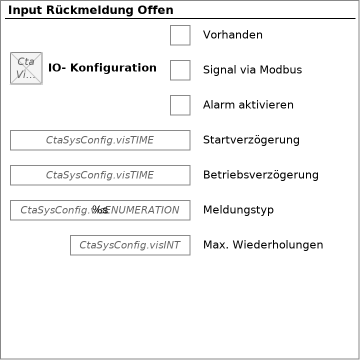
VISUALIZATION StellAntrieb_ParameterIO2  // 360x360
VAR_INPUT
    ITF_STELLANTRIEBIN 	:	ITF_STELLANTRIEB;
	ITF_RückOffen_IN	:	CtaSysIO.ITF_IO;
END_VAR
    Label (5,0 350x20), "Input Rückmeldung Offen"
    Frame (170,25 20x20)
        shows CtaSysConfig.visBOOL(visfbBOOLIn := ITF_STELLANTRIEBIN.p_scInStellAtRükOpen_fbxEnable)
    Label (200,25 150x20), "Vorhanden"
    Frame (170,60 20x20)
        shows CtaSysConfig.visBOOL(visfbBOOLIn := ITF_STELLANTRIEBIN.p_scInStellAtRükOpen_fbxInputMb)
    Label (200,60 150x20), "Signal via Modbus"
    Frame (170,95 20x20)
        shows CtaSysConfig.visBOOL(visfbBOOLIn := ITF_STELLANTRIEBIN.p_scInStellAtRükOpen_fbxDoesAlarm)
    Label (200,95 150x20), "Alarm aktivieren"
    Frame (10,130 180x20)
        shows CtaSysConfig.visTIME(visfbTIMEIn := ITF_STELLANTRIEBIN.p_scInStellAtRükOpen_fbtDelayStart)
    Label (200,130 150x20), "Startverzögerung"
    Label (200,165 150x20), "Betriebsverzögerung"
    Frame (10,165 180x20)
        shows CtaSysConfig.visTIME(visfbTIMEIn := ITF_STELLANTRIEBIN.p_scInStellAtRükOpen_fbtDelayRun)
    Label (200,200 150x20), "Meldungstyp"
    Label (200,235 150x20), "Max. Wiederholungen"
    Line (5,18) (355,18)
    Frame (10,200 180x20)
        shows CtaSysConfig.visENUMERATION(visfbENUIn := ITF_STELLANTRIEBIN.p_scInStellAtRükOpen_fbiTypeOfAck)
    Frame (70,235 120x20)
        shows CtaSysConfig.visINT(visfbINTIn := ITF_STELLANTRIEBIN.p_scInStellAtRükOpen_fbiMaxErrorRetryAllowed)
    Image (10,52 32x32), invisible if: ITF_RückOffen_IN = 0, image: CtaVisSymbols.ImagePool.build
        OnMouseDown:  Dialog=StellAntrieb_POPUP_IO_ITF, Parameters={ITF_IO_IN: ITF_RückOffen_IN}, OpenModal=True, OpenCentered=True
    Label (45,58 120x20), "IO- Konfiguration", invisible if: ITF_RückOffen_IN = 0
    Textfield (30,200 140x20), "%s", text list: 'CtaAppReport.txtLibAp99_2enTypeOfAck', text index: CtaSysConfig.fcGetEnumerationId(ITF_STELLANTRIEBIN.p_scInStellAtRükOpen_fbiTypeOfAck)
END_VISUALIZATION

// 40 Visualizations/POPUP/PARAMETER/StellAntrieb_IO/StellAntrieb_ParameterIO3
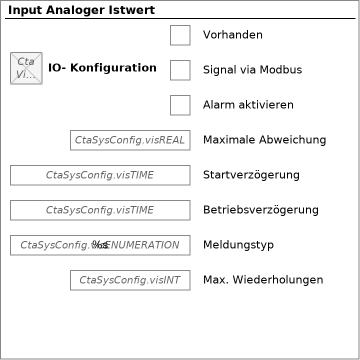
VISUALIZATION StellAntrieb_ParameterIO3  // 360x360
VAR_INPUT
    ITF_STELLANTRIEBIN 	:	ITF_STELLANTRIEB;
	ITF_ActualPos_IN	:	CtaSysIO.ITF_IO;
END_VAR
    Label (5,0 350x20), "Input Analoger Istwert"
    Frame (170,25 20x20)
        shows CtaSysConfig.visBOOL(visfbBOOLIn := ITF_STELLANTRIEBIN.p_scInStellAtActualPosition_fbxEnable)
    Label (200,25 150x20), "Vorhanden"
    Frame (170,60 20x20)
        shows CtaSysConfig.visBOOL(visfbBOOLIn := ITF_STELLANTRIEBIN.p_scInStellAtActualPosition_fbxInputMb)
    Label (200,60 150x20), "Signal via Modbus"
    Frame (170,95 20x20)
        shows CtaSysConfig.visBOOL(visfbBOOLIn := ITF_STELLANTRIEBIN.p_scInStellAtActualPosition_fbxDoesAlarm)
    Label (200,95 150x20), "Alarm aktivieren"
    Frame (10,165 180x20)
        shows CtaSysConfig.visTIME(visfbTIMEIn := ITF_STELLANTRIEBIN.p_scInStellAtActualPosition_fbtDelayStart)
    Label (200,165 150x20), "Startverzögerung"
    Label (200,200 150x20), "Betriebsverzögerung"
    Frame (10,200 180x20)
        shows CtaSysConfig.visTIME(visfbTIMEIn := ITF_STELLANTRIEBIN.p_scInStellAtActualPosition_fbtDelayRun)
    Frame (70,130 120x20)
        shows CtaSysConfig.visREAL(visfbREALIn := ITF_STELLANTRIEBIN.p_scInStellAtActualPosition_fbrMaxDiff, stPhysikalischeEinheit := '%')
    Label (200,130 150x20), "Maximale Abweichung"
    Label (200,235 150x20), "Meldungstyp"
    Label (200,270 150x20), "Max. Wiederholungen"
    Line (5,18) (355,18)
    Frame (10,235 180x20)
        shows CtaSysConfig.visENUMERATION(visfbENUIn := ITF_STELLANTRIEBIN.p_scInStellAtActualPosition_fbiTypeOfAck)
    Frame (70,270 120x20)
        shows CtaSysConfig.visINT(visfbINTIn := ITF_STELLANTRIEBIN.p_scInStellAtActualPosition_fbiMaxErrorRetryAllowed)
    Label (45,58 120x20), "IO- Konfiguration", invisible if: ITF_ActualPos_IN = 0
    Image (10,52 32x32), invisible if: ITF_ActualPos_IN = 0, image: CtaVisSymbols.ImagePool.build
        OnMouseDown:  Dialog=StellAntrieb_POPUP_IO_ITF, Parameters={ITF_IO_IN: ITF_ActualPos_IN}, OpenModal=True, OpenCentered=True
    Textfield (30,235 140x20), "%s", text list: 'CtaAppReport.txtLibAp99_2enTypeOfAck', text index: CtaSysConfig.fcGetEnumerationId(ITF_STELLANTRIEBIN.p_scInStellAtActualPosition_fbiTypeOfAck)
END_VISUALIZATION

// 40 Visualizations/POPUP/PARAMETER/StellAntrieb_InfluxDb/StellAntrieb_ParameterInfluxDb
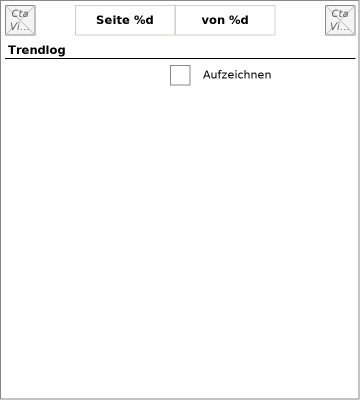
VISUALIZATION StellAntrieb_ParameterInfluxDb  // 360x400
VAR_INPUT
    ITF_STELLANTRIEBIN : ITF_STELLANTRIEB;
END_VAR
VAR
    uiPage  :   UINT;
    uiMin   :   UINT    := 0;
    uiMax   :   UINT    := 0;
END_VAR
    Image (5,5 30x30), invisible if: uiPage = uiMin, image: CtaVisSymbols.ImagePool.arrow-left_square
        OnMouseClick: execute {
            uiPage := uiPage - 1;
            IF uiPage <= uiMin THEN
                uiPage := uiMin;
            END_IF;
        }
    Image (325,5 30x30), invisible if: uiPage = uiMax, image: CtaVisSymbols.ImagePool.arrow-right_square
        OnMouseClick: execute {
            uiPage := uiPage + 1;
            IF uiPage >= uiMax THEN
                uiPage := uiMax;
            END_IF;
        }
    Frame (0,40 360x360), frame switch variable: uiPage
        shows StellAntrieb_ParameterInfluxDb0(ITF_STELLANTRIEBIN := ITF_STELLANTRIEBIN)
        shows AT_ParameterIO1(ITF_Parameter := ITF_Parameter)
        pReferences[0]: ITF_Parameter=ITF_Parameter
    Textfield (75,5 100x30), "Seite %d", text variable: uiPage
    Textfield (175,5 100x30), "von %d", text variable: uiMax
END_VISUALIZATION

// 40 Visualizations/POPUP/PARAMETER/StellAntrieb_InfluxDb/StellAntrieb_ParameterInfluxDb0
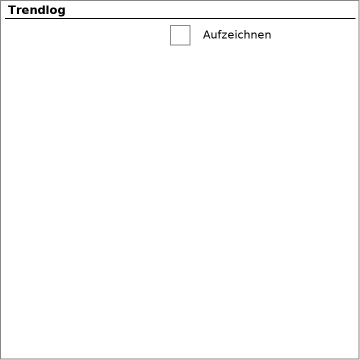
VISUALIZATION StellAntrieb_ParameterInfluxDb0  // 360x360
VAR_INPUT
    ITF_STELLANTRIEBIN : ITF_STELLANTRIEB;
END_VAR
    Frame (170,25 20x20)
        shows CtaSysConfig.visBOOL(visfbBOOLIn := ITF_STELLANTRIEBIN.p_scInfluxDb_fbxEnable)
    Label (200,25 150x20), "Aufzeichnen"
    Label (5,0 350x20), "Trendlog"
    Line (5,18) (355,18)
END_VISUALIZATION

// 40 Visualizations/POPUP/IO/StellAntrieb_IO0
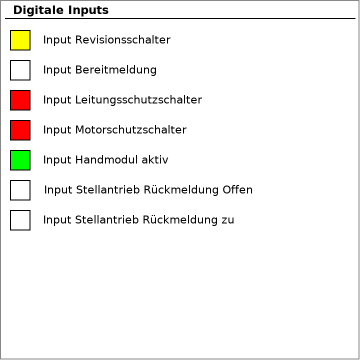
VISUALIZATION StellAntrieb_IO0  // 360x360
VAR_INPUT
    ITF_STELLANTRIEBIN    :   ITF_STELLANTRIEB;	
END_VAR
    Label (40,30 320x20), "Input Revisionsschalter", invisible if: ITF_STELLANTRIEBIN.proNotShowDI_RevisionSwitchOk
    Label (40,60 320x20), "Input Bereitmeldung", invisible if: ITF_STELLANTRIEBIN.proNotShowDI_Ready
    Rectangle (10,30 20x20), colour toggle: ITF_STELLANTRIEBIN.proGetDI_RevisionSwitchOK, invisible if: ITF_STELLANTRIEBIN.proNotShowDI_RevisionSwitchOk
    Rectangle (10,60 20x20), colour toggle: ITF_STELLANTRIEBIN.proGetDI_IsReady, invisible if: ITF_STELLANTRIEBIN.proNotShowDI_Ready
    Rectangle (10,90 20x20), colour toggle: ITF_STELLANTRIEBIN.proGetDI_FuseOK, invisible if: ITF_STELLANTRIEBIN.proNotShowDI_FuseOk
    Label (40,90 320x20), "Input Leitungsschutzschalter", invisible if: ITF_STELLANTRIEBIN.proNotShowDI_FuseOk
    Label (40,120 320x20), "Input Motorschutzschalter", invisible if: ITF_STELLANTRIEBIN.proNotShowDI_ActuatorFuseOk
    Rectangle (10,120 20x20), colour toggle: ITF_STELLANTRIEBIN.proGetDI_ActuatorFuseOk, invisible if: ITF_STELLANTRIEBIN.proNotShowDI_ActuatorFuseOk
    Label (40,150 320x20), "Input Handmodul aktiv", invisible if: ITF_STELLANTRIEBIN.proNotShowDI_ActuatorHand
    Rectangle (10,150 20x20), colour toggle: ITF_STELLANTRIEBIN.proGetDI_ActuatorHand, invisible if: ITF_STELLANTRIEBIN.proNotShowDI_ActuatorHand
    Label (10,0 350x20), "Digitale Inputs"
    Rectangle (10,210 20x20), colour toggle: ITF_STELLANTRIEBIN.proGetDI_RükIsClosed, invisible if: ITF_STELLANTRIEBIN.proNotShowDI_RükIsOpen
    Label (40,210 320x20), "Input Stellantrieb Rückmeldung zu", invisible if: ITF_STELLANTRIEBIN.proNotShowDI_RükIsOpen
    Rectangle (10,180 20x20), colour toggle: ITF_STELLANTRIEBIN.proGetDI_RükIsOpen, invisible if: ITF_STELLANTRIEBIN.proNotShowDI_RükIsOpen
    Label (41,180 320x20), "Input Stellantrieb Rückmeldung Offen", invisible if: ITF_STELLANTRIEBIN.proNotShowDI_RükIsOpen
    Line (5,18) (355,18)
END_VISUALIZATION

// 40 Visualizations/POPUP/IO/StellAntrieb_IO
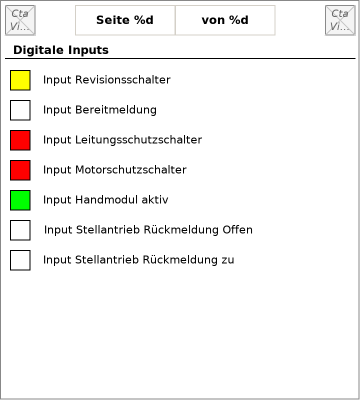
VISUALIZATION StellAntrieb_IO  // 360x400
VAR_INPUT
    ITF_STELLANTRIEBIN    :   ITF_STELLANTRIEB;	
END_VAR
VAR
    uiPage  :   UINT;
    uiMin   :   UINT    := 0;
    uiMax   :   UINT    := 1;
END_VAR
    Frame (0,40 360x360), frame switch variable: uiPage
        shows StellAntrieb_IO0(ITF_STELLANTRIEBIN := ITF_STELLANTRIEBIN)
        shows StellAntrieb_IO1(ITF_STELLANTRIEBIN := ITF_STELLANTRIEBIN)
        shows AT_ParameterIO2(ITF_Parameter := ITF_Parameter)
        shows AT_ParameterIO3(ITF_Parameter := ITF_Parameter)
    Image (325,5 30x30), invisible if: uiPage = uiMax, image: CtaVisSymbols.ImagePool.arrow-right_square
        OnMouseClick: execute {
            uiPage := uiPage + 1;
            IF uiPage >= uiMax THEN
                uiPage := uiMax;
            END_IF;
        }
    Image (5,5 30x30), invisible if: uiPage = uiMin, image: CtaVisSymbols.ImagePool.arrow-left_square
        OnMouseClick: execute {
            uiPage := uiPage - 1;
            IF uiPage <= uiMin THEN
                uiPage := uiMin;
            END_IF;
        }
    Textfield (175,5 100x30), "von %d", text variable: uiMax
    Textfield (75,5 100x30), "Seite %d", text variable: uiPage
END_VISUALIZATION

// 40 Visualizations/POPUP/IO/StellAntrieb_IO1
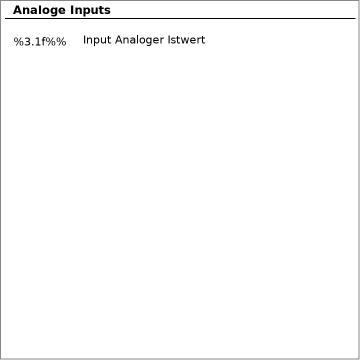
VISUALIZATION StellAntrieb_IO1  // 360x360
VAR_INPUT
    ITF_STELLANTRIEBIN    :   ITF_STELLANTRIEB;	
END_VAR
    Label (80,30 280x20), "Input Analoger Istwert", invisible if: ITF_STELLANTRIEBIN.proNotShowAI_ActualPosition
    Label (10,0 350x20), "Analoge Inputs"
    Textfield (10,32 60x20), "%3.1f%%", text variable: ITF_STELLANTRIEBIN.proGetAI_ActualPosition, invisible if: ITF_STELLANTRIEBIN.proNotShowAI_ActualPosition
    Line (5,18) (355,18)
END_VISUALIZATION

// 40 Visualizations/ICON/StellAntrieb_BASE/Ventile/DurchflussVentil/Motor_Left/ML_Durchgang
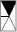
VISUALIZATION ML_Durchgang  // 17x32
VAR_INPUT
	rProzent	:	REAL;
END_VAR
VAR
	A			:	fbValveAnimation := (CenterPoint0 := (iX := 9, iY := 16),Direction := 1,SquareDimension := 15);
END_VAR
    Line (1,16) (9,16)
    Polygon (9,16) (16,1) (1,1)
    Polygon (9,16) (16,31) (1,31)
    Polygon (9,16) (16,1) (1,1)
        p1285906596: A.CalculatePolygon(rProzent,TRUE)
END_VISUALIZATION

// 40 Visualizations/ICON/StellAntrieb_BASE/Icons/Motor_Left/Icon_ML_AB_Down
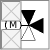
VISUALIZATION Icon_ML_AB_Down  // 50x50
VAR_INPUT
    ITF_STELLANTRIEB_IN   :   ITF_STELLANTRIEB;	
END_VAR
    Frame (4,16 18x18)
        shows Motor(ITF_STELLANTRIEB_IN := ITF_STELLANTRIEB_IN)
    Frame (20,9 24x32)
        shows ML_Ventil_AB_Down(rProzent := ITF_STELLANTRIEB_IN.proOnY)
    Image (1,1 20x20), invisible if: NOT ITF_STELLANTRIEB_IN.proIsWarning, image: CtaVisSymbols.ImagePool.CtaWarning
    Image (1,29 20x20), invisible if: NOT ITF_STELLANTRIEB_IN.proIsHandOnOrOff, image: CtaVisSymbols.ImagePool.front_hand_Yellow
    Image (1,29 20x20), invisible if: NOT ITF_STELLANTRIEB_IN.proHandOff, image: CtaVisSymbols.ImagePool.front_hand_Yellow_Off
END_VISUALIZATION

// 40 Visualizations/ICON/StellAntrieb_BASE/Ventile/DreiWegVentil/Motor_Above/MA_Ventil_AB_L
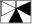
VISUALIZATION MA_Ventil_AB_L  // 32x24
VAR_INPUT
	rProzent	:	REAL;
END_VAR
VAR
	A			:	fbValveAnimation := (CenterPoint0 := (iX := 16, iY := 8),Direction := 2,SquareDimension := 15);
	B			:	fbValveAnimation := (CenterPoint0 := (iX := 16, iY := 8),Direction := 0,SquareDimension := 15);
END_VAR
    Polygon (1,1) (16,8) (1,16)
    Polygon (16,8) (23,23) (8,23)
    Polygon (16,8) (31,1) (31,16)
    Line (16,8) (16,1)
    Polygon (16,8) (31,1) (31,16)
        p1285906596: A.CalculatePolygon(rProzent,TRUE)
    Polygon (16,8) (23,23) (8,23)
        p1285906596: B.CalculatePolygon(rProzent,FALSE)
END_VISUALIZATION

// 40 Visualizations/ICON/StellAntrieb_BASE/Ventile/DreiWegVentil/Motor_Above/MA_Ventil_Verteiler
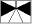
VISUALIZATION MA_Ventil_Verteiler  // 32x24
VAR_INPUT
	rProzent	:	REAL;
END_VAR
VAR
	A			:	fbValveAnimation := (CenterPoint0 := (iX := 16, iY := 8),Direction := 3,SquareDimension := 15);
	B			:	fbValveAnimation := (CenterPoint0 := (iX := 16, iY := 8),Direction := 2,SquareDimension := 15);
END_VAR
    Polygon (1,1) (16,8) (1,16)
    Polygon (16,8) (23,23) (8,23)
    Polygon (16,8) (31,1) (31,16)
    Line (16,8) (16,1)
    Polygon (16,8) (31,1) (31,16)
        p1285906596: B.CalculatePolygon(rProzent,FALSE)
    Polygon (1,1) (16,8) (1,16)
        p1285906596: A.CalculatePolygon(rProzent,TRUE)
END_VISUALIZATION

// 40 Visualizations/ICON/StellAntrieb_BASE/Ventile/DreiWegVentil/Motor_Above/MA_Ventil_AB_R
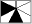
VISUALIZATION MA_Ventil_AB_R  // 32x24
VAR_INPUT
	rProzent	:	REAL;
END_VAR
VAR
	A			:	fbValveAnimation := (CenterPoint0 := (iX := 16, iY := 8),Direction := 3,SquareDimension := 15);
	B			:	fbValveAnimation := (CenterPoint0 := (iX := 16, iY := 8),Direction := 0,SquareDimension := 15);
END_VAR
    Polygon (1,1) (16,8) (1,16)
    Polygon (16,8) (23,23) (8,23)
    Polygon (16,8) (31,1) (31,16)
    Line (16,8) (16,1)
    Polygon (16,8) (23,23) (8,23)
        p1285906596: B.CalculatePolygon(rProzent,FALSE)
    Polygon (1,1) (16,8) (1,16)
        p1285906596: A.CalculatePolygon(rProzent,TRUE)
END_VISUALIZATION

// 40 Visualizations/ICON/StellAntrieb_BASE/Ventile/DreiWegVentil/Motor_Left/ML_Ventil_AB_Down
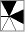
VISUALIZATION ML_Ventil_AB_Down  // 25x32
VAR_INPUT
	rProzent	:	REAL;
END_VAR
VAR
	A			:	fbValveAnimation := (CenterPoint0 := (iX := 9, iY := 16),Direction := 1,SquareDimension := 15);
	B			:	fbValveAnimation := (CenterPoint0 := (iX := 9, iY := 16),Direction := 2,SquareDimension := 15);
END_VAR
    Polygon (9,16) (16,1) (1,1)
    Polygon (9,16) (16,31) (1,31)
    Polygon (9,16) (24,9) (24,24)
    Line (1,16) (10,16)
    Polygon (9,16) (24,9) (24,24)
        p1285906596: B.CalculatePolygon(rProzent,FALSE)
    Polygon (9,16) (16,1) (1,1)
        p1285906596: A.CalculatePolygon(rProzent,TRUE)
END_VISUALIZATION

// 40 Visualizations/ICON/StellAntrieb_BASE/Ventile/DreiWegVentil/Motor_Left/ML_Ventil_Verteiler
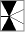
VISUALIZATION ML_Ventil_Verteiler  // 25x32
VAR_INPUT
	rProzent	:	REAL;
END_VAR
VAR
	A			:	fbValveAnimation := (CenterPoint0 := (iX := 9, iY := 16),Direction := 0,SquareDimension := 15);
	B			:	fbValveAnimation := (CenterPoint0 := (iX := 9, iY := 16),Direction := 1,SquareDimension := 15);
END_VAR
    Polygon (9,16) (16,1) (1,1)
    Polygon (9,16) (16,31) (1,31)
    Polygon (9,16) (24,9) (24,24)
    Line (1,16) (10,16)
    Polygon (9,16) (16,1) (1,1)
        p1285906596: B.CalculatePolygon(rProzent,FALSE)
    Polygon (9,16) (16,31) (1,31)
        p1285906596: A.CalculatePolygon(rProzent,TRUE)
END_VISUALIZATION

// 40 Visualizations/ICON/StellAntrieb_BASE/Ventile/DreiWegVentil/Motor_Left/ML_Ventil_AB_Up
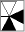
VISUALIZATION ML_Ventil_AB_Up  // 25x32
VAR_INPUT
	rProzent	:	REAL;
END_VAR
VAR
	A			:	fbValveAnimation := (CenterPoint0 := (iX := 9, iY := 16),Direction := 0,SquareDimension := 15);
	B			:	fbValveAnimation := (CenterPoint0 := (iX := 9, iY := 16),Direction := 2,SquareDimension := 15);
END_VAR
    Polygon (9,16) (16,1) (1,1)
    Polygon (9,16) (16,31) (1,31)
    Polygon (9,16) (24,9) (24,24)
    Line (1,16) (10,16)
    Polygon (9,16) (24,9) (24,24)
        p1285906596: B.CalculatePolygon(rProzent,FALSE)
    Polygon (9,16) (16,31) (1,31)
        p1285906596: A.CalculatePolygon(rProzent,TRUE)
END_VISUALIZATION

// 40 Visualizations/ICON/StellAntrieb_BASE/Ventile/DreiWegVentil/Motor_Below/MB_Ventil_AB_L
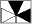
VISUALIZATION MB_Ventil_AB_L  // 32x24
VAR_INPUT
	rProzent	:	REAL;
END_VAR
VAR
	A			:	fbValveAnimation := (CenterPoint0 := (iX := 16, iY := 16),Direction := 2,SquareDimension := 15);
	B			:	fbValveAnimation := (CenterPoint0 := (iX := 16, iY := 16),Direction := 1,SquareDimension := 15);
END_VAR
    Polygon (16,16) (23,1) (8,1)
    Polygon (1,8) (16,15) (1,23)
    Polygon (16,15) (31,8) (31,23)
    Line (16,23) (16,14)
    Polygon (16,15) (31,8) (31,23)
        p1285906596: A.CalculatePolygon(rProzent,TRUE)
    Polygon (16,15) (23,1) (8,1)
        p1285906596: B.CalculatePolygon(rProzent,FALSE)
END_VISUALIZATION

// 40 Visualizations/ICON/StellAntrieb_BASE/Ventile/DreiWegVentil/Motor_Below/MB_Ventil_Verteiler
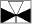
VISUALIZATION MB_Ventil_Verteiler  // 32x24
VAR_INPUT
	rProzent	:	REAL;
END_VAR
VAR
	A			:	fbValveAnimation := (CenterPoint0 := (iX := 16, iY := 16),Direction := 3,SquareDimension := 15);
	B			:	fbValveAnimation := (CenterPoint0 := (iX := 16, iY := 16),Direction := 2,SquareDimension := 15);
END_VAR
    Polygon (16,16) (23,1) (8,1)
    Polygon (1,8) (16,15) (1,23)
    Polygon (16,15) (31,8) (31,23)
    Line (16,23) (16,14)
    Polygon (16,15) (31,8) (31,23)
        p1285906596: B.CalculatePolygon(rProzent,TRUE)
    Polygon (1,8) (16,15) (1,23)
        p1285906596: A.CalculatePolygon(rProzent,FALSE)
END_VISUALIZATION

// 40 Visualizations/ICON/StellAntrieb_BASE/Ventile/DreiWegVentil/Motor_Below/MB_Ventil_AB_R
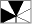
VISUALIZATION MB_Ventil_AB_R  // 32x24
VAR_INPUT
	rProzent	:	REAL;
END_VAR
VAR
	A			:	fbValveAnimation := (CenterPoint0 := (iX := 16, iY := 16),Direction := 3,SquareDimension := 15);
	B			:	fbValveAnimation := (CenterPoint0 := (iX := 16, iY := 16),Direction := 1,SquareDimension := 15);
END_VAR
    Polygon (16,16) (23,1) (8,1)
    Polygon (1,8) (16,16) (1,23)
    Polygon (16,16) (31,8) (31,23)
    Line (16,23) (16,14)
    Polygon (16,16) (1,8) (1,23)
        p1285906596: A.CalculatePolygon(rProzent,TRUE)
    Polygon (16,16) (23,1) (8,1)
        p1285906596: B.CalculatePolygon(rProzent,FALSE)
END_VISUALIZATION

// 40 Visualizations/ICON/StellAntrieb_BASE/Ventile/DreiWegVentil/Motor_Right/MR_Ventil_AB_Up
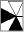
VISUALIZATION MR_Ventil_AB_Up  // 24x32
VAR_INPUT
	rProzent	:	REAL;
END_VAR
VAR
	A			:	fbValveAnimation := (CenterPoint0 := (iX := 16, iY := 16),Direction := 0,SquareDimension := 15);
	B			:	fbValveAnimation := (CenterPoint0 := (iX := 16, iY := 16),Direction := 3,SquareDimension := 15);
END_VAR
    Polygon (16,16) (23,1) (8,1)
    Polygon (16,16) (23,31) (8,31)
    Polygon (16,16) (1,8) (1,23)
    Line (15,16) (23,16)
    Polygon (16,16) (1,8) (1,23)
        p1285906596: B.CalculatePolygon(rProzent,FALSE)
    Polygon (16,16) (23,31) (8,31)
        p1285906596: A.CalculatePolygon(rProzent,TRUE)
END_VISUALIZATION

// 40 Visualizations/ICON/StellAntrieb_BASE/Ventile/DreiWegVentil/Motor_Right/MR_Ventil_Verteiler
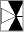
VISUALIZATION MR_Ventil_Verteiler  // 24x32
VAR_INPUT
	rProzent	:	REAL;
END_VAR
VAR
	A			:	fbValveAnimation := (CenterPoint0 := (iX := 16, iY := 16),Direction := 1,SquareDimension := 15);
	B			:	fbValveAnimation := (CenterPoint0 := (iX := 16, iY := 16),Direction := 0,SquareDimension := 15);
END_VAR
    Polygon (16,16) (23,1) (8,1)
    Polygon (16,16) (23,31) (8,31)
    Polygon (16,16) (1,8) (1,23)
    Line (15,16) (23,16)
    Polygon (16,16) (23,1) (8,1)
        p1285906596: A.CalculatePolygon(rProzent,FALSE)
    Polygon (16,16) (23,31) (8,31)
        p1285906596: B.CalculatePolygon(rProzent,TRUE)
END_VISUALIZATION

// 40 Visualizations/ICON/StellAntrieb_BASE/Ventile/DreiWegVentil/Motor_Right/MR_Ventil_AB_Down
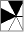
VISUALIZATION MR_Ventil_AB_Down  // 24x32
VAR_INPUT
	rProzent	:	REAL;
END_VAR
VAR
	A			:	fbValveAnimation := (CenterPoint0 := (iX := 16, iY := 16),Direction := 1,SquareDimension := 15);
	B			:	fbValveAnimation := (CenterPoint0 := (iX := 16, iY := 16),Direction := 3,SquareDimension := 15);
END_VAR
    Polygon (16,16) (23,1) (8,1)
    Polygon (16,16) (23,31) (8,31)
    Polygon (16,16) (1,8) (1,23)
    Line (15,16) (23,16)
    Polygon (16,16) (23,1) (8,1)
        p1285906596: A.CalculatePolygon(rProzent,FALSE)
    Polygon (16,16) (1,8) (1,23)
        p1285906596: B.CalculatePolygon(rProzent,TRUE)
END_VISUALIZATION

// 40 Visualizations/ICON/StellAntrieb_BASE/Ventile/DurchflussVentil/Motor_Right/MR_Durchgang
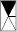
VISUALIZATION MR_Durchgang  // 17x32
VAR_INPUT
	rProzent	:	REAL;
END_VAR
VAR
	A			:	fbValveAnimation := (CenterPoint0 := (iX := 8, iY := 16),Direction := 1,SquareDimension := 15);
END_VAR
    Line (8,16) (16,16)
    Polygon (8,16) (16,1) (1,1)
    Polygon (8,16) (16,31) (1,31)
    Polygon (8,16) (16,1) (1,1)
        p1285906596: A.CalculatePolygon(rProzent,TRUE)
END_VISUALIZATION

// 40 Visualizations/ICON/StellAntrieb_BASE/Ventile/DurchflussVentil/Motor_Below/MB_Durchgang
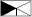
VISUALIZATION MB_Durchgang  // 32x17
VAR_INPUT
	rProzent	:	REAL;
END_VAR
VAR
	A			:	fbValveAnimation := (CenterPoint0 := (iX := 16, iY := 9),Direction := 3,SquareDimension := 15);
END_VAR
    Line (16,8) (16,16)
    Polygon (1,1) (16,8) (1,16)
    Polygon (16,8) (31,1) (31,16)
    Polygon (1,1) (16,8) (1,16)
        p1285906596: A.CalculatePolygon(rProzent,TRUE)
END_VISUALIZATION

// 40 Visualizations/ICON/StellAntrieb_BASE/Ventile/DurchflussVentil/Motor_Above/MA_Durchgang
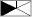
VISUALIZATION MA_Durchgang  // 32x17
VAR_INPUT
	rProzent	:	REAL;
END_VAR
VAR
	A			:	fbValveAnimation := (CenterPoint0 := (iX := 16, iY := 8),Direction := 3,SquareDimension := 15);
END_VAR
    Line (16,1) (16,8)
    Polygon (1,1) (16,8) (1,16)
    Polygon (16,8) (31,1) (31,16)
    Polygon (1,1) (16,8) (1,16)
        p1285906596: A.CalculatePolygon(rProzent,TRUE)
END_VISUALIZATION

// 40 Visualizations/ICON/StellAntrieb_BASE/Icons/Motor_Left/Icon_ML_AB_Up
